// TIA Portal V20 export
TYPE "LER_typeEmRelationEm_05"
// stored: Access Published, Namespace Unit1
   STRUCT
      commonBit : Array[0..99] of Bool;
      commonInt : Array[0..10] of Int;
      leftBit : Array[0..99] of Bool;
      rightBit : Array[0..99] of Bool;
      leftInt : Array[0..99] of Int;
      rightInt : Array[0..99] of Int;
      leftPartData : "LER_typePartData";
      rightPartData : "LER_typePartData";
      homeCheck : Array[0..199] of Bool;
      homed : Array[0..31] of Bool;
      axis : Array[0..31] of Struct
         interlock : Array[0..99] of Bool;
         inposDone : Array[0..99] of Bool;
         inposDoneBefore : Array[0..99] of Bool;
         inposDoneAfter : Array[0..99] of Bool;
         Moving : Array[0..99] of Bool;
      END_STRUCT;
      cylinder : Array[0..31] of Struct
         inHomePosInterlock : Bool;
         inWorkPosInterlock : Bool;
         inHomePosDone : Bool;
         inWorkPosDone : Bool;
      END_STRUCT;
      digitalSignal : Array[0..31] of Bool;
      leftLoading : Struct
         request : Array[0..63] of Bool;
         ready : Array[0..63] of Bool;
         done : Array[0..63] of Bool;
      END_STRUCT;
      rightLoading : Struct
         request : Array[0..63] of Bool;
         ready : Array[0..63] of Bool;
         done : Array[0..63] of Bool;
      END_STRUCT;
      leftUnloading : Struct
         request : Array[0..63] of Bool;
         ready : Array[0..63] of Bool;
         done : Array[0..63] of Bool;
      END_STRUCT;
      rightUnloading : Struct
         request : Array[0..63] of Bool;
         ready : Array[0..63] of Bool;
         done : Array[0..63] of Bool;
      END_STRUCT;
      leftClamp : Struct
         request : Array[0..63] of Bool;
         ready : Array[0..63] of Bool;
         done : Array[0..63] of Bool;
      END_STRUCT;
      rightClamp : Struct
         request : Array[0..63] of Bool;
         ready : Array[0..63] of Bool;
         done : Array[0..63] of Bool;
      END_STRUCT;
      leftUnclamp : Struct
         request : Array[0..63] of Bool;
         ready : Array[0..63] of Bool;
         done : Array[0..63] of Bool;
      END_STRUCT;
      rightUnclamp : Struct
         request : Array[0..63] of Bool;
         ready : Array[0..63] of Bool;
         done : Array[0..63] of Bool;
      END_STRUCT;
      leftWorking : Struct
         ready : Array[0..63] of Bool;
         done : Array[0..63] of Bool;
      END_STRUCT;
      rightWorking : Struct
         ready : Array[0..63] of Bool;
         done : Array[0..63] of Bool;
      END_STRUCT;
      sequence : Array[0..9] of Struct
         job : Array[0..99] of Struct
            locked : Bool;
            active : Bool;
            completed : Bool;
            aborted : Bool;
         END_STRUCT;
      END_STRUCT;
      "r&r" : Struct
         thickness : Struct
            select : Bool;
            workingDone : Bool;
         END_STRUCT;
         vision : Struct
            select : Bool;
            workingDone : Bool;
         END_STRUCT;
         weight : Struct
            select : Bool;
            workingDone : Bool;
         END_STRUCT;
      END_STRUCT;
      axisEnabled_DR14 : Bool;
      axisEnabled_DR17 : Bool;
   END_STRUCT;
END_TYPE
